// TIA Portal V21 export
DATA_BLOCK "Vessel_Lamp"   // DB1
// stored: AutoNumber false, InstanceOfName TIMER, InstanceOfType FB
"TIMER"
   // VAR_INPUT
   //    TIME_START : Bool;
   //    TIME_PULSE : Bool;
   //    TIME_TRSET : Bool;
   //    MINI_ENABLE : Bool;
   //    TIME_IN_MINI : DInt;
   //    TIME_IN_SEC : DInt;
   // END_VAR
   // VAR_OUTPUT
   //    DONE_BIT : Bool;
   //    ES_MINIT : DInt;
   //    ES_SEC : DInt;
   // END_VAR
   // VAR_IN_OUT
   //    TEMP_1 : DInt;
   //    TEMP_5 : DInt;
   //    TEMP_2 : DInt;
   //    TEMP_3 : DInt;
   //    TEMP_BIT_1 : Bool;
   //    TEMP_BIT_2 : Bool;
   // END_VAR
BEGIN
END_DATA_BLOCK
